SUBAPPLICATION Tageszaehler (* Subapplication Type *)
  (* Standard: 61499-2 *)
  (* Version 1.0, 2023-02-17, Franz *)
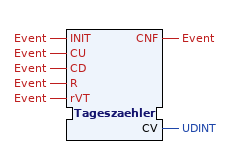
  EVENT_INPUT
    INIT; (* Initialization Request *)
    CU; (* Count Up *)
    CD; (* Count Down *)
    R; (* Reset *)
    rVT; (* refresh VT *)
  END_EVENT
  EVENT_OUTPUT
    CNF; (* Confirmation -- Counter Value was changed *)
  END_EVENT
  VAR_OUTPUT
    CV : UDINT; (* Counter Value *)
  END_VAR
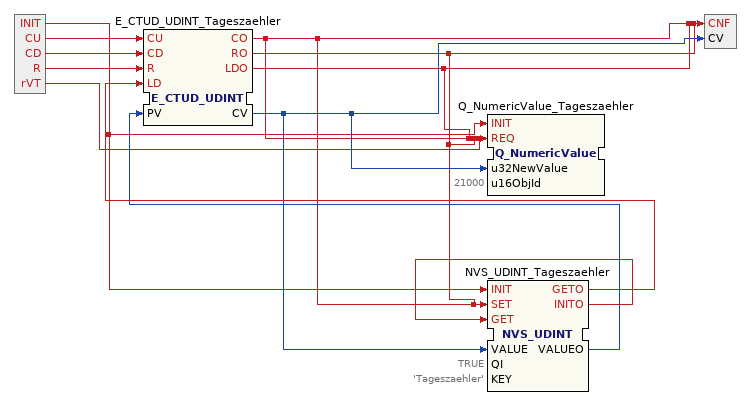
  FBS
    E_CTUD_UDINT_Tageszaehler : E_CTUD_UDINT;
    Q_NumericValue_Tageszaehler : Q_NumericValue(u16ObjId := 21000);
    NVS_UDINT_Tageszaehler : NVS_UDINT(QI := TRUE, KEY := 'Tageszaehler');
  END_FBS
  EVENT_CONNECTIONS
    INIT TO Q_NumericValue_Tageszaehler.INIT;
    E_CTUD_UDINT_Tageszaehler.CO TO Q_NumericValue_Tageszaehler.REQ;
    E_CTUD_UDINT_Tageszaehler.RO TO Q_NumericValue_Tageszaehler.REQ;
    E_CTUD_UDINT_Tageszaehler.LDO TO Q_NumericValue_Tageszaehler.REQ;
    CU TO E_CTUD_UDINT_Tageszaehler.CU;
    CD TO E_CTUD_UDINT_Tageszaehler.CD;
    R TO E_CTUD_UDINT_Tageszaehler.R;
    INIT TO NVS_UDINT_Tageszaehler.INIT;
    E_CTUD_UDINT_Tageszaehler.CO TO NVS_UDINT_Tageszaehler.SET;
    E_CTUD_UDINT_Tageszaehler.RO TO NVS_UDINT_Tageszaehler.SET;
    NVS_UDINT_Tageszaehler.GETO TO E_CTUD_UDINT_Tageszaehler.LD;
    NVS_UDINT_Tageszaehler.INITO TO NVS_UDINT_Tageszaehler.GET;
    E_CTUD_UDINT_Tageszaehler.CO TO CNF;
    E_CTUD_UDINT_Tageszaehler.RO TO CNF;
    E_CTUD_UDINT_Tageszaehler.LDO TO CNF;
    rVT TO Q_NumericValue_Tageszaehler.REQ;
  END_CONNECTIONS
  DATA_CONNECTIONS
    E_CTUD_UDINT_Tageszaehler.CV TO Q_NumericValue_Tageszaehler.u32NewValue;
    E_CTUD_UDINT_Tageszaehler.CV TO NVS_UDINT_Tageszaehler.VALUE;
    NVS_UDINT_Tageszaehler.VALUEO TO E_CTUD_UDINT_Tageszaehler.PV;
    E_CTUD_UDINT_Tageszaehler.CV TO CV;
  END_CONNECTIONS
END_SUBAPPLICATION
